TYPE ST_LPTTS_State :
STRUCT
	// LoadPort module state , 2 LPs
	arrLoadPort: ARRAY [1..(.NO_OF_LPS)] OF ST_LPState;
	// TTS moduel state
	stTTS: ST_TTS_State;
		
END_STRUCT
END_TYPE

(* stored: Version 1.1.0.1, ProductVersion 3.1.4022.12
   DUT ST_LPTTS_State: Id {5ab772ee-5e76-4d92-af29-4b436d405b07} *)
